PROGRAM Water_Tank
VAR
	start:BOOL;
	stop:BOOL;
	high:BOOL;
	low:BOOL;
	motor:BOOL;
	temp:BOOL;
	mix:BOOL;
	release:BOOL;
	
	TON_0: TON;
	TOF_0: TOF;
	TON_1: TON;
	MixFor10S: TOF;
	Delay2S: TON;
END_VAR

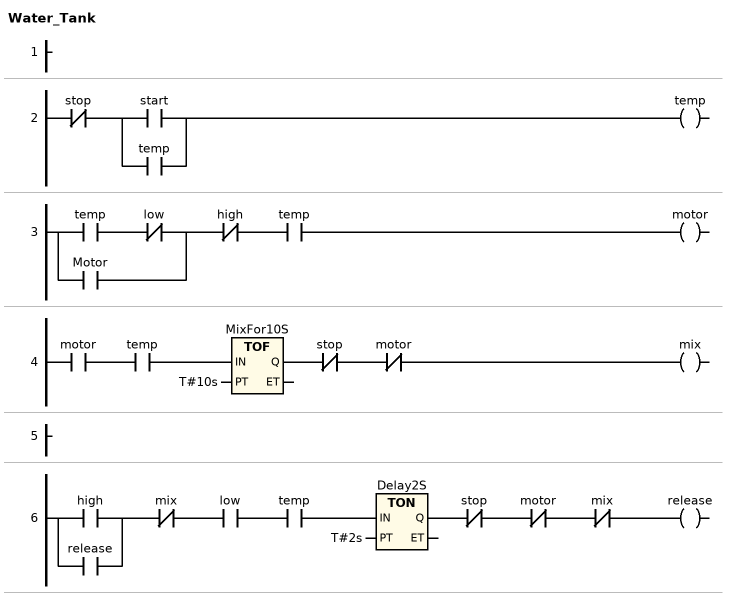
// NETWORK 1

// NETWORK 2
temp := NOT stop AND (start OR temp);

// NETWORK 3
motor := (temp AND NOT low OR Motor) AND NOT high AND temp;

// NETWORK 4
MixFor10S(IN := motor AND temp, PT := T#10s); // TOF
mix := MixFor10S.Q AND NOT stop AND NOT motor;

// NETWORK 5

// NETWORK 6
Delay2S(IN := (high OR release) AND NOT mix AND low AND temp, PT := T#2s); // TON
release := Delay2S.Q AND NOT stop AND NOT motor AND NOT mix;

END_PROGRAM

(* stored: Version 1.1.0.1, ProductVersion 3.1.4024.12
   POU Water_Tank: Id {c8021f2c-e80b-41ce-aed7-000ec211807f}, SpecialFunc None *)
